{attribute 'linkalways'} 
{attribute 'no_explicit_call' := 'This FB is a CLASS and must be accessed using methods or properties'}
{attribute 'enable_dynamic_creation'}
FUNCTION_BLOCK Table IMPLEMENTS I_Table
VAR
	_fb : FB_NciFeedTablePreparation;
	_table : ST_NciFeedGroupTable;
	
	_stopped : STRING;
	_errorId : UDINT;
	_filledRows : INT;
END_VAR

PROPERTY _InternalTable : REFERENCE TO Tc2_PlcInterpolation.ST_NciFeedGroupTable
GET
_InternalTable REF= _table;
END_GET
END_PROPERTY

METHOD AddAxisDynamics : BOOL
VAR_INPUT
	displayIndex : UDINT;
	axis : mobject_motion.I_Axis;
	acceleration : LREAL(0.000001-99999999);
	deceleration : LREAL(0.000001-99999999);
	jerk : LREAL(0.000001-99999999);
END_VAR
VAR
	entry : ST_NciAxisDynamics;
END_VAR
entry.nDisplayIndex := displayIndex;
entry.nAxis := axis.AxisId;
entry.fAcc := acceleration;
entry.fDec := deceleration;
entry.fJerk := jerk;

_fb(
	stFeedGroupTable := _table,
	pEntry := ADR(entry),
	nEntryType := Tc2_PlcInterpolation.E_NciEntryType.E_NciEntryTypeAxisDynamics,
	bResetTable := FALSE,
	bResetAll := FALSE,
	nFilledRows => _filledRows
);

AddAxisDynamics := _fb.bError;
END_METHOD

METHOD AddBaseFrame : BOOL
VAR_INPUT
	displayIndex : UDINT;
	shiftX : LREAL;
	shiftY : LREAL;
	shiftZ : LREAL;
	rotationX : LREAL;
	rotationY : LREAL;
	rotationZ : LREAL;
	shiftQ1 : LREAL;
	shiftQ2 : LREAL;
	shiftQ3 : LREAL;
	shiftQ4 : LREAL;
	shiftQ5 : LREAL;
END_VAR
VAR
	entry : ST_NciBaseFrame;
END_VAR
entry.nDisplayIndex := displayIndex;
entry.fShiftX := shiftX;
entry.fShiftY := shiftY;
entry.fShiftZ := shiftZ;
entry.fRotX := rotationX;
entry.fRotY := rotationY;
entry.fRotZ := rotationZ;
entry.fShiftQ1 := shiftQ1;
entry.fShiftQ2 := shiftQ2;
entry.fShiftQ3 := shiftQ3;
entry.fShiftQ4 := shiftQ4;
entry.fShiftQ5 := shiftQ5;

_fb(
	stFeedGroupTable := _table,
	pEntry := ADR(entry),
	nEntryType := Tc2_PlcInterpolation.E_NciEntryType.E_NciEntryTypeBaseFrame,
	bResetTable := FALSE,
	bResetAll := FALSE,
	nFilledRows => _filledRows
);

AddBaseFrame := _fb.bError;
END_METHOD

METHOD AddBaseFrame3D : BOOL
VAR_INPUT
	displayIndex : UDINT;
	shiftX : LREAL;
	shiftY : LREAL;
	shiftZ : LREAL;
	rotationX : LREAL;
	rotationY : LREAL;
	rotationZ : LREAL;
END_VAR
AddBaseFrame3D := AddBaseFrame(
	displayIndex,
	shiftX, shiftY, shiftZ,
	rotationX, rotationY, rotationZ,
	0, 0, 0, 0, 0
);
END_METHOD

METHOD AddBezier3rdOrder : BOOL
VAR_INPUT
	displayIndex : UDINT;
	controlPoint1X : LREAL;
	controlPoint1Y : LREAL;
	controlPoint1Z : LREAL;
	controlPoint2X : LREAL;
	controlPoint2Y : LREAL;
	controlPoint2Z : LREAL;
	endPositionX : LREAL;
	endPositionY : LREAL;
	endPositionZ : LREAL;
	endPositionQ1 : LREAL;
	endPositionQ2 : LREAL;
	endPositionQ3 : LREAL;
	endPositionQ4 : LREAL;
	endPositionQ5 : LREAL;
	velocity : LREAL(0.000001-99999999);
	accurateStop : BOOL; // velocity at end == 0
END_VAR
VAR
	entry : ST_NciGeoBezier3;
END_VAR
entry.nDisplayIndex := displayIndex;
entry.fControlPoint1X := controlPoint1X;
entry.fControlPoint1Y := controlPoint1Y;
entry.fControlPoint1Z := controlPoint1Z;
entry.fControlPoint2X := controlPoint2X;
entry.fControlPoint2Y := controlPoint2Y;
entry.fControlPoint2Z := controlPoint2Z;
entry.fEndPosX := endPositionX;
entry.fEndPosY := endPositionY;
entry.fEndPosZ := endPositionZ;
entry.fEndPosQ1 := endPositionQ1;
entry.fEndPosQ2 := endPositionQ2;
entry.fEndPosQ3 := endPositionQ3;
entry.fEndPosQ4 := endPositionQ4;
entry.fEndPosQ5 := endPositionQ5;
entry.fVelo := velocity;
entry.bAccurateStop := accurateStop;

_fb(
	stFeedGroupTable := _table,
	pEntry := ADR(entry),
	nEntryType := Tc2_PlcInterpolation.E_NciEntryType.E_NciEntryTypeGeoBezier3,
	bResetTable := FALSE,
	bResetAll := FALSE,
	nFilledRows => _filledRows
);

AddBezier3rdOrder := _fb.bError;
END_METHOD

METHOD AddBezier3rdOrder3D : BOOL
VAR_INPUT
	displayIndex : UDINT;
	controlPoint1X : LREAL;
	controlPoint1Y : LREAL;
	controlPoint1Z : LREAL;
	controlPoint2X : LREAL;
	controlPoint2Y : LREAL;
	controlPoint2Z : LREAL;
	endPositionX : LREAL;
	endPositionY : LREAL;
	endPositionZ : LREAL;
	velocity : LREAL(0.000001-99999999);
	accurateStop : BOOL; // velocity at end == 0
END_VAR
AddBezier3rdOrder3D := AddBezier3rdOrder(
	displayIndex,
	controlPoint1X, controlPoint1Y, controlPoint1Z,
	controlPoint2X, controlPoint2Y, controlPoint2Z,
	endPositionX, endPositionY, endPositionZ,
	0, 0, 0, 0, 0,
	velocity,
	accurateStop
);
END_METHOD

METHOD AddBezier5thOrder : BOOL
VAR_INPUT
	displayIndex : UDINT;
	controlPoint1X : LREAL;
	controlPoint1Y : LREAL;
	controlPoint1Z : LREAL;
	controlPoint2X : LREAL;
	controlPoint2Y : LREAL;
	controlPoint2Z : LREAL;
	controlPoint3X : LREAL;
	controlPoint3Y : LREAL;
	controlPoint3Z : LREAL;
	controlPoint4X : LREAL;
	controlPoint4Y : LREAL;
	controlPoint4Z : LREAL;
	endPositionX : LREAL;
	endPositionY : LREAL;
	endPositionZ : LREAL;
	endPositionQ1 : LREAL;
	endPositionQ2 : LREAL;
	endPositionQ3 : LREAL;
	endPositionQ4 : LREAL;
	endPositionQ5 : LREAL;
	velocity : LREAL(0.000001-99999999);
	accurateStop : BOOL; // velocity at end == 0
END_VAR
VAR
	entry : ST_NciGeoBezier5;
END_VAR
entry.nDisplayIndex := displayIndex;
entry.fControlPoint1X := controlPoint1X;
entry.fControlPoint1Y := controlPoint1Y;
entry.fControlPoint1Z := controlPoint1Z;
entry.fControlPoint2X := controlPoint2X;
entry.fControlPoint2Y := controlPoint2Y;
entry.fControlPoint2Z := controlPoint2Z;
entry.fControlPoint3X := controlPoint3X;
entry.fControlPoint3Y := controlPoint3Y;
entry.fControlPoint3Z := controlPoint3Z;
entry.fControlPoint4X := controlPoint4X;
entry.fControlPoint4Y := controlPoint4Y;
entry.fControlPoint4Z := controlPoint4Z;
entry.fEndPosX := endPositionX;
entry.fEndPosY := endPositionY;
entry.fEndPosZ := endPositionZ;
entry.fEndPosQ1 := endPositionQ1;
entry.fEndPosQ2 := endPositionQ2;
entry.fEndPosQ3 := endPositionQ3;
entry.fEndPosQ4 := endPositionQ4;
entry.fEndPosQ5 := endPositionQ5;
entry.fVelo := velocity;
entry.bAccurateStop := accurateStop;

_fb(
	stFeedGroupTable := _table,
	pEntry := ADR(entry),
	nEntryType := Tc2_PlcInterpolation.E_NciEntryType.E_NciEntryTypeGeoBezier5,
	bResetTable := FALSE,
	bResetAll := FALSE,
	nFilledRows => _filledRows
);

AddBezier5thOrder := _fb.bError;
END_METHOD

METHOD AddBezier5thOrder3D : BOOL
VAR_INPUT
	displayIndex : UDINT;
	controlPoint1X : LREAL;
	controlPoint1Y : LREAL;
	controlPoint1Z : LREAL;
	controlPoint2X : LREAL;
	controlPoint2Y : LREAL;
	controlPoint2Z : LREAL;
	controlPoint3X : LREAL;
	controlPoint3Y : LREAL;
	controlPoint3Z : LREAL;
	controlPoint4X : LREAL;
	controlPoint4Y : LREAL;
	controlPoint4Z : LREAL;
	endPositionX : LREAL;
	endPositionY : LREAL;
	endPositionZ : LREAL;
	velocity : LREAL(0.000001-99999999);
	accurateStop : BOOL; // velocity at end == 0
END_VAR
AddBezier5thOrder3D := AddBezier5thOrder(
	displayIndex,
	controlPoint1X, controlPoint1Y, controlPoint1Z,
	controlPoint2X, controlPoint2Y, controlPoint2Z,
	controlPoint3X, controlPoint3Y, controlPoint3Z,
	controlPoint4X, controlPoint4Y, controlPoint4Z,
	endPositionX, endPositionY, endPositionZ,
	0, 0, 0, 0, 0,
	velocity,
	accurateStop
);
END_METHOD

METHOD AddCircleCIP : BOOL
VAR_INPUT
	displayIndex : UDINT;
	endPositionX : LREAL;
	endPositionY : LREAL;
	endPositionZ : LREAL;
	arcPointX : LREAL;
	arcPointY : LREAL;
	arcPointZ : LREAL;
	endPositionQ1 : LREAL;
	endPositionQ2 : LREAL;
	endPositionQ3 : LREAL;
	endPositionQ4 : LREAL;
	endPositionQ5 : LREAL;
	velocity : LREAL(0.000001-99999999);
	accurateStop : BOOL; // velocity at end == 0
END_VAR
VAR
	entry : ST_NciGeoCircleCIP;
END_VAR
entry.nDisplayIndex := displayIndex;
entry.fEndPosX := endPositionX;
entry.fEndPosY := endPositionY;
entry.fEndPosZ := endPositionZ;
entry.fCIPPosX := arcPointX;
entry.fCIPPosY := arcPointY;
entry.fCIPPosZ := arcPointZ;
entry.fEndPosQ1 := endPositionQ1;
entry.fEndPosQ2 := endPositionQ2;
entry.fEndPosQ3 := endPositionQ3;
entry.fEndPosQ4 := endPositionQ4;
entry.fEndPosQ5 := endPositionQ5;
entry.fVelo := velocity;
entry.bAccurateStop := accurateStop;

_fb(
	stFeedGroupTable := _table,
	pEntry := ADR(entry),
	nEntryType := Tc2_PlcInterpolation.E_NciEntryType.E_NciEntryTypeGeoCircleCIP,
	bResetTable := FALSE,
	bResetAll := FALSE,
	nFilledRows => _filledRows
);

AddCircleCIP := _fb.bError;
END_METHOD

METHOD AddCircleCIP3D : BOOL
VAR_INPUT
	displayIndex : UDINT;
	endPositionX : LREAL;
	endPositionY : LREAL;
	endPositionZ : LREAL;
	arcPointX : LREAL;
	arcPointY : LREAL;
	arcPointZ : LREAL;
	velocity : LREAL(0.000001-99999999);
	accurateStop : BOOL; // velocity at end == 0
END_VAR
AddCircleCIP3D := AddCircleCIP(
	displayIndex,
	endPositionX, endPositionY, endPositionZ,
	arcPointX, arcPointY, arcPointZ,
	0, 0, 0, 0, 0,
	velocity,
	accurateStop
);
END_METHOD

METHOD AddCircleOnPlane : BOOL
VAR_INPUT
	displayIndex : UDINT;
	endPositionX : LREAL;
	endPositionY : LREAL;
	endPositionZ : LREAL;
	centerX : LREAL;
	centerY : LREAL;
	centerZ : LREAL;
	endPositionQ1 : LREAL;
	endPositionQ2 : LREAL;
	endPositionQ3 : LREAL;
	endPositionQ4 : LREAL;
	endPositionQ5 : LREAL;
	plane : StandardPlane := StandardPlane.XY;
	clockwise : BOOL;	
	velocity : LREAL(0.000001-99999999);
	accurateStop : BOOL; // velocity at end == 0
END_VAR
VAR
	entry: ST_NciGeoCirclePlane;
END_VAR
entry.nDisplayIndex := displayIndex;
entry.fEndPosX := endPositionX;
entry.fEndPosY := endPositionY;
entry.fEndPosZ := endPositionZ;
entry.fCenterX := centerX;
entry.fCenterY := centerY;
entry.fCenterZ := centerZ;
entry.fEndPosQ1 := endPositionQ1;
entry.fEndPosQ2 := endPositionQ2;
entry.fEndPosQ3 := endPositionQ3;
entry.fEndPosQ4 := endPositionQ4;
entry.fEndPosQ5 := endPositionQ5;
entry.nPlane := plane;
entry.bClockwise := clockwise;
entry.fVelo := velocity;
entry.bAccurateStop := accurateStop;

_fb(
	stFeedGroupTable := _table,
	pEntry := ADR(entry),
	nEntryType := Tc2_PlcInterpolation.E_NciEntryType.E_NciEntryTypeGeoCirclePlane,
	bResetTable := FALSE,
	bResetAll := FALSE,
	nFilledRows => _filledRows
);

AddCircleOnPlane := _fb.bError;
END_METHOD

METHOD AddCircleOnPlane3D : BOOL
VAR_INPUT
	displayIndex : UDINT;
	endPositionX : LREAL;
	endPositionY : LREAL;
	endPositionZ : LREAL;
	centerX : LREAL;
	centerY : LREAL;
	centerZ : LREAL;
	plane : StandardPlane := StandardPlane.XY;
	clockwise : BOOL;
	velocity : LREAL(0.000001-99999999);
	accurateStop : BOOL; // velocity at end == 0
END_VAR
AddCircleOnPlane3D := AddCircleOnPlane(
	displayIndex,
	endPositionX,
	endPositionY,
	endPositionZ,
	centerX ,
	centerY,
	centerZ,
	0, 0, 0, 0, 0,
	plane,
	clockwise,	
	velocity,
	accurateStop
);
END_METHOD

METHOD AddDwellTime : BOOL
VAR_INPUT
	displayIndex : UDINT;
	dwellTime : LREAL(0.000001-99999999); // seconds
END_VAR
VAR
	entry: ST_NciDwellTime;
END_VAR
entry.nDisplayIndex := displayIndex;
entry.fDwellTime := dwellTime;

_fb(
	stFeedGroupTable := _table,
	pEntry := ADR(entry),
	nEntryType := Tc2_PlcInterpolation.E_NciEntryType.E_NciEntryTypeDwellTime,
	bResetTable := FALSE,
	bResetAll := FALSE,
	nFilledRows => _filledRows
);

AddDwellTime := _fb.bError;
END_METHOD

METHOD AddFeedrateInterpolation : BOOL
VAR_INPUT
	displayIndex : UDINT;
	interpolationType : FeedrateInterpolation;
END_VAR
VAR
	entry : ST_NciFeedrateIpol;
END_VAR
entry.nDisplayIndex := displayIndex;
entry.eFeedrateIpol := interpolationType;

_fb(
	stFeedGroupTable := _table,
	pEntry := ADR(entry),
	nEntryType := Tc2_PlcInterpolation.E_NciEntryType.E_NciEntryTypeFeedrateIpol,
	bResetTable := FALSE,
	bResetAll := FALSE,
	nFilledRows => _filledRows
);

 AddFeedrateInterpolation:= _fb.bError;
END_METHOD

METHOD AddLine : BOOL
VAR_INPUT
	displayIndex : UDINT;
	endPositionX : LREAL;
	endPositionY : LREAL;
	endPositionZ : LREAL;
	endPositionQ1 : LREAL;
	endPositionQ2 : LREAL;
	endPositionQ3 : LREAL;
	endPositionQ4 : LREAL;
	endPositionQ5 : LREAL;
	velocity : LREAL(0.000001-99999999);
	rapidTraverse : BOOL;
	accurateStop : BOOL; // velocity at end == 0
END_VAR
VAR
	entry : ST_NciGeoLine;
END_VAR
entry.nDisplayIndex := displayIndex;
entry.fEndPosX := endPositionX;
entry.fEndPosY := endPositionY;
entry.fEndPosZ := endPositionZ;
entry.fEndPosQ1 := endPositionQ1;
entry.fEndPosQ2 := endPositionQ2;
entry.fEndPosQ3 := endPositionQ3;
entry.fEndPosQ4 := endPositionQ4;
entry.fEndPosQ5 := endPositionQ5;
entry.fVelo := velocity;
entry.bRapidTraverse := rapidTraverse;
entry.bAccurateStop := accurateStop;

_fb(
	stFeedGroupTable := _table,
	pEntry := ADR(entry),
	nEntryType := Tc2_PlcInterpolation.E_NciEntryType.E_NciEntryTypeGeoLine,
	bResetTable := FALSE,
	bResetAll := FALSE,
	nFilledRows => _filledRows
);

AddLine := _fb.bError;
END_METHOD

METHOD AddLine3D : BOOL
VAR_INPUT
	displayIndex : UDINT;
	endPositionX : LREAL;
	endPositionY : LREAL;
	endPositionZ : LREAL;
	velocity : LREAL(0.000001-99999999);
	rapidTraverse : BOOL;
	accurateStop : BOOL; // velocity at end == 0
END_VAR
AddLine3D := AddLine(
	displayIndex,
	endPositionX,
	endPositionY,
	endPositionZ,
	0, 0, 0, 0, 0,
	velocity,
	rapidTraverse,
	accurateStop
);
END_METHOD

METHOD AddMFunctionWithHandshake : BOOL
VAR_INPUT
	displayIndex : UDINT;
	functionNumber : INT(0..159);
END_VAR
VAR
	entry : ST_NciMFuncHsk;
END_VAR
entry.nDisplayIndex := displayIndex;
entry.nMFunc := functionNumber;

_fb(
	stFeedGroupTable := _table,
	pEntry := ADR(entry),
	nEntryType := Tc2_PlcInterpolation.E_NciEntryType.E_NciEntryTypeMFuncHsk,
	bResetTable := FALSE,
	bResetAll := FALSE,
	nFilledRows => _filledRows
);

 AddMFunctionWithHandshake := _fb.bError;
END_METHOD

METHOD AddPathDynamics : BOOL
VAR_INPUT
	displayIndex : UDINT;
	acceleration : LREAL(0.000001-99999999);
	deceleration : LREAL(0.000001-99999999);
	jerk : LREAL(0.000001-99999999);
END_VAR
VAR
	entry : ST_NciPathDynamics;
END_VAR
entry.nDisplayIndex := displayIndex;
entry.fAcc := acceleration;
entry.fDec := deceleration;
entry.fJerk := jerk;

_fb(
	stFeedGroupTable := _table,
	pEntry := ADR(entry),
	nEntryType := Tc2_PlcInterpolation.E_NciEntryType.E_NciEntryTypePathDynamics,
	bResetTable := FALSE,
	bResetAll := FALSE,
	nFilledRows => _filledRows
);

AddPathDynamics := _fb.bError;
END_METHOD

METHOD AddReference
END_METHOD

METHOD AddStart : BOOL
VAR_INPUT
	x : LREAL;
	y : LREAL;
	z : LREAL;
	q1 : LREAL;
	q2 : LREAL;
	q3 : LREAL;
	q4 : LREAL;
	q5 : LREAL;
END_VAR
VAR
	entry : ST_NciGeoStart;
END_VAR
entry.fPosX := x;
entry.fPosY := y;
entry.fPosZ := z;
entry.fPosQ1 := q1;
entry.fPosQ2 := q2;
entry.fPosQ3 := q3;
entry.fPosQ4 := q4;
entry.fPosQ5 := q5;

_fb(
	stFeedGroupTable := _table,
	pEntry := ADR(entry),
	nEntryType := Tc2_PlcInterpolation.E_NciEntryType.E_NciEntryTypeGeoStart,
	bResetTable := FALSE,
	bResetAll := FALSE,
	nFilledRows => _filledRows
);

AddStart := _fb.bError;
END_METHOD

METHOD AddStart3D : BOOL
VAR_INPUT
	x : LREAL;
	y : LREAL;
	z : LREAL;
END_VAR
AddStart3D := AddStart(x, y, z, 0, 0, 0, 0, 0);
END_METHOD

METHOD DisableTangentialFollowing : BOOL
VAR
	entry : ST_NciTangentialFollowingDesc;
END_VAR
entry.bTangOn := FALSE;

_fb(
	stFeedGroupTable := _table,
	pEntry := ADR(entry),
	nEntryType := Tc2_PlcInterpolation.E_NciEntryType.E_NciEntryTypeTfDesc,
	bResetTable := FALSE,
	bResetAll := FALSE,
	nFilledRows => _filledRows
);

DisableTangentialFollowing := _fb.bError;
END_METHOD

METHOD DisableVertexSmoothing : BOOL
VAR_INPUT
	displayIndex : UDINT;
END_VAR
DisableVertexSmoothing := EnableVertexSmoothing(
	displayIndex,
	VertexSmoothingBlendingType.NONE,
	VertexSmoothingSubType.NONE,
	0
);
END_METHOD

METHOD EnableTangentialFollowing : BOOL
VAR_INPUT
	tangentialAxis : NciAxis; // axis used for tangential following
	pathAxis1 : NciAxis; // describing the plane e.g. x
	pathAxis2 : NciAxis; // e.g. y ==> g17, xy plane
	offset : LREAL; // geo tangent is 0 degree, counting is mathmatical positive
	criticalAngle : LREAL(0.000001-90);
	behaviour : TangentialFollowingBehaviour;
END_VAR
VAR
	entry : ST_NciTangentialFollowingDesc;
END_VAR
entry.bTangOn := TRUE;
entry.nTangAxis := tangentialAxis;
entry.nPathAxis1 := pathAxis1;
entry.nPathAxis2 := pathAxis2;
entry.fOffset := offset;
entry.fCriticalAngle1 := criticalAngle;
entry.nTfBehavior := behaviour;

_fb(
	stFeedGroupTable := _table,
	pEntry := ADR(entry),
	nEntryType := Tc2_PlcInterpolation.E_NciEntryType.E_NciEntryTypeTfDesc,
	bResetTable := FALSE,
	bResetAll := FALSE,
	nFilledRows => _filledRows
);

EnableTangentialFollowing := _fb.bError;
END_METHOD

METHOD EnableVertexSmoothing : BOOL
VAR_INPUT
	displayIndex : UDINT;
	blendType : VertexSmoothingBlendingType;
	subType : VertexSmoothingSubType;
	radius : LREAL(0.000001-99999999);
END_VAR
VAR
	entry : ST_NciVertexSmoothing;
END_VAR
entry.nEntryType := Tc2_PlcInterpolation.E_NciEntryType.E_NciEntryTypeVertexSmoothing;
entry.nDisplayIndex := displayIndex;
entry.nType := blendType;
entry.nSubtype :=	subType;
entry.fRadius :=	radius;

_fb(
	stFeedGroupTable := _table,
	pEntry := ADR(entry),
	nEntryType := Tc2_PlcInterpolation.E_NciEntryType.E_NciEntryTypeVertexSmoothing,
	bResetTable := FALSE,
	bResetAll := FALSE,
	nFilledRows => _filledRows
);

EnableVertexSmoothing := _fb.bError;
END_METHOD

METHOD End : BOOL
VAR
	entry : ST_NciEndOfTables;
END_VAR
_fb(
	stFeedGroupTable := _table,
	pEntry := ADR(entry),
	nEntryType := Tc2_PlcInterpolation.E_NciEntryType.E_NciEntryTypeEndOfTables,
	bResetTable := FALSE,
	bResetAll := FALSE,
	nFilledRows => _filledRows
);

End := _fb.bError;
END_METHOD

PROPERTY ErrorId : UDINT
GET
ErrorId := _fb.nErrorId;
END_GET
END_PROPERTY

PROPERTY FilledRows : INT
GET
FilledRows := _filledRows;
END_GET
END_PROPERTY

PROPERTY HasError : BOOL
GET
HasError := _fb.bError;
END_GET
END_PROPERTY

METHOD ResetAll : BOOL
_fb(
	stFeedGroupTable := _table,
	bResetAll := TRUE
);

ResetAll := _fb.bError;
END_METHOD

METHOD ResetTable : BOOL
_fb(
	stFeedGroupTable := _table,
	bResetTable := TRUE
);

ResetTable := _fb.bError;
END_METHOD

END_FUNCTION_BLOCK

(* stored: Version 1.1.0.1, ProductVersion 3.1.4024.12
   POU Table: Id {59162d18-0ee0-4cf5-a92a-47a2b71f5b59}, SpecialFunc None
   Property _InternalTable: Id {58136a9d-fe87-4a07-86bf-28af7e84c4d0}
   Get Get: Id {c802491e-4974-4916-9c66-579775e4f6a4}
   Method AddAxisDynamics: Id {c9b688c8-c844-4a2a-aac1-e47eec851813}
   Method AddBaseFrame: Id {2d830661-64a0-4be4-b0ce-ae13155622a1}
   Method AddBaseFrame3D: Id {1b840118-50a3-4dba-ac58-e7bc5fe05011}
   Method AddBezier3rdOrder: Id {d5f88368-fb96-4702-ada4-647eda08d402}
   Method AddBezier3rdOrder3D: Id {90533534-41d5-4b8f-9a47-4920a8bba202}
   Method AddBezier5thOrder: Id {768fcc9d-d1c2-47a5-bab0-0b773ea03856}
   Method AddBezier5thOrder3D: Id {6c695a21-d481-4b70-91e1-da433a8f6892}
   Method AddCircleCIP: Id {1993b774-ee2a-4084-bf57-ba803bb6351a}
   Method AddCircleCIP3D: Id {16a132ac-edd2-4a86-9c0e-a5bdd7ca3c4b}
   Method AddCircleOnPlane: Id {ab9e2afb-4da1-4459-b464-aa1953da5d04}
   Method AddCircleOnPlane3D: Id {4d29e5ba-7892-413f-ae85-e5c601974f36}
   Method AddDwellTime: Id {85506703-5108-460a-8ae3-29d5b1eb0b12}
   Method AddFeedrateInterpolation: Id {abfd7b6c-2d57-4aa0-b541-20f14bcb430e}
   Method AddLine: Id {6af79330-da5a-4362-a3e9-c4e02127b9a9}
   Method AddLine3D: Id {b3962469-8f0b-4933-bbf4-cea7aa6e5ee2}
   Method AddMFunctionWithHandshake: Id {ea5b16be-5020-4eee-9e51-8e4eb9c2d10f}
   Method AddPathDynamics: Id {bf0a7c94-cf1a-4f10-8493-ec901c65bc72}
   Method AddReference: Id {bf3eac9d-5726-4886-a224-eb9105cbbb87}
   Method AddStart: Id {0aff247d-c14b-4817-9473-d4eddbd39da2}
   Method AddStart3D: Id {2a090461-743e-4da8-8eea-88c674e929ac}
   Method DisableTangentialFollowing: Id {0e53d2d8-efd3-4d67-8206-d874cf816509}
   Method DisableVertexSmoothing: Id {60412a89-ef33-4113-82e1-ed369327ddb9}
   Method EnableTangentialFollowing: Id {bc04643a-92a6-4acd-aaee-0f429c0d86f2}
   Method EnableVertexSmoothing: Id {d1118b77-a80d-4547-b16b-6b195fb3f946}
   Method End: Id {2f3f9392-649b-452d-b693-fac8229271ae}
   Property ErrorId: Id {f4e1beb3-2a39-4700-a39b-04ba09f8778e}
   Get Get: Id {105dc9bd-2ae2-44c7-8274-48ba52853a02}
   Property FilledRows: Id {6cbd3997-07bc-4187-9c61-7ae082c7a13e}
   Get Get: Id {6ae5f1dc-7657-4da4-bb46-c40fa1301377}
   Property HasError: Id {87e36c8a-94a2-49fb-b284-1d79850c966e}
   Get Get: Id {8ab7970f-c403-4e73-b592-aba4e50c4ed6}
   Method ResetAll: Id {55fddf7a-e7ea-4752-adc5-0cbbc94290b7}
   Method ResetTable: Id {53b82f7d-fa9f-4577-ac9c-22ccd621f88f} *)
